{attribute addProperty BoxType "EL6201-0000-0017"}
{attribute addProperty Id "Slave_6A_DI0BIT10.12541Slave_6A_DI1BIT10.12542Slave_6A_DI2BIT10.12543Slave_6A_DI3BIT10.12544Slave_6B_DI0BIT10.12545Slave_6B_DI1BIT10.12546Slave_6B_DI2BIT10.12547Slave_6B_DI3BIT10.12548"}
{attribute addProperty CRC "1066543944"}
{attribute addProperty SizeInBites "8"}
{attribute addProperty SizeInBytes "1"}
TYPE Slave_6_Inputs_3F922B48 :
STRUCT
	{attribute addProperty Name "Slave_6A_DI0"}
	Slave_6A_DI0 : BIT;
	{attribute addProperty Name "Slave_6A_DI1"}
	Slave_6A_DI1 : BIT;
	{attribute addProperty Name "Slave_6A_DI2"}
	Slave_6A_DI2 : BIT;
	{attribute addProperty Name "Slave_6A_DI3"}
	Slave_6A_DI3 : BIT;
	{attribute addProperty Name "Slave_6B_DI0"}
	Slave_6B_DI0 : BIT;
	{attribute addProperty Name "Slave_6B_DI1"}
	Slave_6B_DI1 : BIT;
	{attribute addProperty Name "Slave_6B_DI2"}
	Slave_6B_DI2 : BIT;
	{attribute addProperty Name "Slave_6B_DI3"}
	Slave_6B_DI3 : BIT;
END_STRUCT
END_TYPE

(* stored: Version 1.2.0.0, ProductVersion 3.1.4024.9
   DUT Slave_6_Inputs_3F922B48: Id {a7ecbead-492b-4ad7-b43f-a61a63b2333a} *)
